// TIA Portal V20 export
// export: Created 2026-04-11T06:02:30.6791533Z, ExportSetting WithDefaults, DisplayName Totally Integrated Automation Portal, DisplayVersion V20, DisplayName TIA Portal Openness, DisplayVersion V20, DisplayName TIA Portal Version Control Interface, DisplayVersion V20, DisplayName STEP 7 Professional, DisplayVersion V20, DisplayName STEP 7 Safety, DisplayVersion V20, DisplayName WinCC Basic/Comfort/Advanced, DisplayVersion V20, DisplayName WinCC Unified, DisplayVersion V20
TYPE "udtHMI_PID_Config"
// stored: IsFailsafeCompliant false
   STRUCT
      rGainP : Real;
      rGainI : Real;
      rGainD : Real;
      rIntegralErrorThreshold : Real;
      rOutputMin : Real;
      rOutputMax : Real;
      rDerivativeFilterWeight : Real;
      rDisabledOutput : Real;
      bReverseActing : Bool;
   END_STRUCT;
END_TYPE
